// TIA Portal project "trafficLight_timer_counter" (V16)

(* hardware
DEVICE "S7-1200 station_1"  S7-1200 Station
   slot 0: "Rack_0"  S7-1200 Rack  Rack  V1.0
   slot 1: "PLC_1"  CPU 1214C DC/DC/DC  6ES7 214-1AG40-0XB0  V4.4
DEVICE "HMI_1"  KTP700 Basic PN
   slot 0: "HMI_1"  KTP700 Basic PN  6AV2 123-2GB03-0AX0  16.0.0.0
   slot 1: "HMI_RT_1"  KTP700 Basic PN  6AV2 123-2GB03-0AX0  16.0.0.0
   slot 5: "HMI_1.IE_CP_1"  PROFINET Interface  16.0.0.0
      slot 1: "PROFINET Interface_1"  PROFINET Interface
         slot 1: "Port_1"  Port
*)

// ===== PLC "PLC_1"  CPU 1214C DC/DC/DC =====

VAR_GLOBAL   // PLC tag table "Default tag table"
   "GREENTON" AT %MD10 : Time;
   "START(1)" AT %Q0.4 : Bool;
   "RED_SEM" AT %Q0.0 : Bool;
   "REDTON" AT %MD18 : Time;
   "GREEN_SEM" AT %Q0.2 : Bool;
   "BLUETON" AT %MD14 : Time;
   "BLUETON_SEM" AT %MD16 : Time;
   "Tag_8" AT %MD22 : Time;
   "Tag_9" AT %I0.0 : Bool;
   "START(2)" AT %I0.1 : Bool;
   "Tag_11" AT %I0.5 : Bool;
   "STOP_SEM" AT %I1.0 : Bool;
   "BLUE_SEM" AT %Q0.1 : Bool;
   "VALVULA" AT %Q0.3 : Bool;
   "START_SEM" AT %I0.4 : Bool;
   "MEMORIA0" AT %M0.0 : Bool;
   "MEMORIA0.1" AT %M0.1 : Bool;
   "Tag_1" AT %M0.2 : Bool;
   "Tag_3" AT %MW50 : Word;
   "STOP" AT %Q1.0 : Bool;
   "value_norm_x1" AT %IW64 : Int;
   "out_norm_x1" AT %MD200 : Real;
   "value_scale_x1" AT %MD100 : Real;
   "PRESION_VALUE_REAL_scalex1" AT %MD104 : Real;
   "Tag_2" AT %IW68 : Int;
   "Tag_4" AT %MW208 : Word;
   "Tag_5" AT %MD208 : Real;
   "Tag_6" AT %MD102 : Real;
   "Tag_10" AT %MD108 : Real;
   "Tag_12" AT %MD112 : Real;
   "GREENTON_SEM" AT %MD12 : Time;
   "REDTON_SEM" AT %MD20 : Time;
END_VAR

// folder: System blocks/Program resources

DATA_BLOCK "TON1"   // DB2
{ S7_Optimized_Access := 'TRUE' }
AUTHOR : Simatic
FAMILY : IEC
NAME : IEC_TMR
VERSION : 1.0
// stored: InstanceOfName IEC_TIMER
"IEC_TIMER"
BEGIN
END_DATA_BLOCK

DATA_BLOCK "TON2"   // DB5
{ S7_Optimized_Access := 'TRUE' }
AUTHOR : Simatic
FAMILY : IEC
NAME : IEC_TMR
VERSION : 1.0
// stored: InstanceOfName IEC_TIMER
"IEC_TIMER"
BEGIN
END_DATA_BLOCK

DATA_BLOCK "CTU1"   // DB8
{ S7_Optimized_Access := 'TRUE' }
AUTHOR : Simatic
FAMILY : IEC
NAME : CNTR
VERSION : 1.0
// stored: InstanceOfName IEC_COUNTER
"IEC_COUNTER"
BEGIN
END_DATA_BLOCK

DATA_BLOCK "TON3"   // DB10
{ S7_Optimized_Access := 'TRUE' }
AUTHOR : Simatic
FAMILY : IEC
NAME : IEC_TMR
VERSION : 1.0
// stored: InstanceOfName IEC_TIMER
"IEC_TIMER"
BEGIN
END_DATA_BLOCK

// folder: (top level)

FUNCTION "SEMAFORO" : Void   // FC2, LAD
{ S7_Optimized_Access := 'TRUE' }
VERSION : 0.1
BEGIN

REGION Network 1
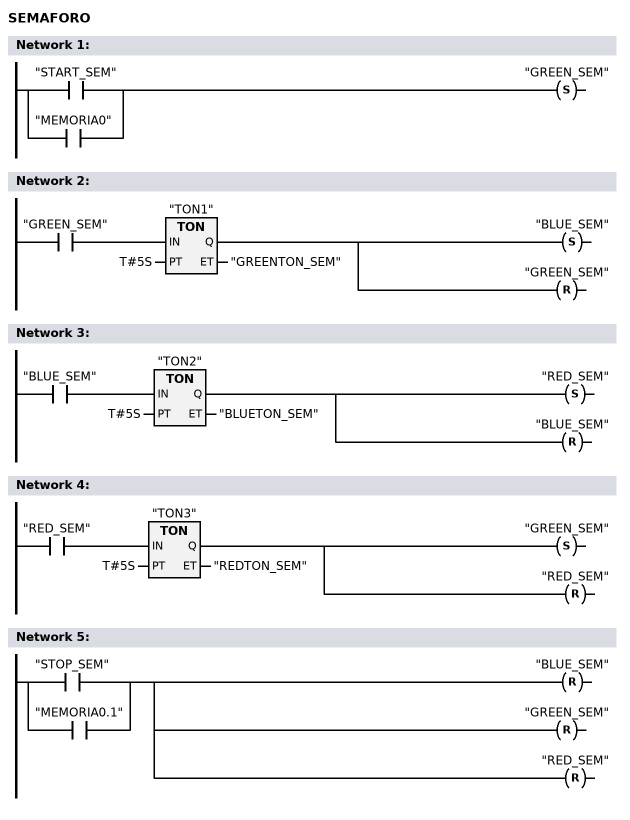
   RUNG wire#powerrail
      Contact( "START_SEM" )
      wire#w1
      S_Coil( "GREEN_SEM" )
   END_RUNG
   RUNG wire#powerrail
      Contact( "MEMORIA0" )
   END_RUNG wire#w1
   // the same network as SCL:
   IF "START_SEM" OR "MEMORIA0" THEN "GREEN_SEM" := TRUE; END_IF;
END_REGION

REGION Network 2
   "TON1".TON(IN := "GREEN_SEM", PT := T#5S, ET => "GREENTON_SEM");
   IF "TON1".Q THEN
       "BLUE_SEM" := TRUE;
       "GREEN_SEM" := FALSE;
   END_IF;
END_REGION

REGION Network 3
   "TON2".TON(IN := "BLUE_SEM", PT := T#5S, ET => "BLUETON_SEM");
   IF "TON2".Q THEN
       "RED_SEM" := TRUE;
       "BLUE_SEM" := FALSE;
   END_IF;
END_REGION

REGION Network 4
   "TON3".TON(IN := "RED_SEM", PT := T#5S, ET => "REDTON_SEM");
   IF "TON3".Q THEN
       "GREEN_SEM" := TRUE;
       "RED_SEM" := FALSE;
   END_IF;
END_REGION

REGION Network 5
   RUNG wire#powerrail
      Contact( "STOP_SEM" )
      wire#w1
      R_Coil( "BLUE_SEM" )
   END_RUNG
   RUNG wire#powerrail
      Contact( "MEMORIA0.1" )
   END_RUNG wire#w1
   RUNG wire#w1
      R_Coil( "GREEN_SEM" )
   END_RUNG
   RUNG wire#w1
      R_Coil( "RED_SEM" )
   END_RUNG
   // the same network as SCL:
   IF "STOP_SEM" OR "MEMORIA0.1" THEN
       "BLUE_SEM" := FALSE;
       "GREEN_SEM" := FALSE;
       "RED_SEM" := FALSE;
   END_IF;
END_REGION
END_FUNCTION

FUNCTION "CONTADOR" : Void   // FC3, LAD
{ S7_Optimized_Access := 'TRUE' }
VERSION : 0.1
   VAR_TEMP   // added for the SCL form of the ladder/FBD networks
      _w1 : Bool;
   END_VAR
BEGIN

REGION Network 1: CONTADOR CTU SIMPLE CON FLANCO DE BAJADA
   // PROHIBICION DE PARTNER OBJECT ELECCION EN SUS PARAMETROS : en memory N item
   // LIMITES CANTIDAD DE ELECCION EN SUS PARAMETROS
   // N ES DE FLANCO DE BAJADAAA
   // si pv = 3, el contador empieza en 0 y se incrementa de 1 en 1 hasta llegar a 3
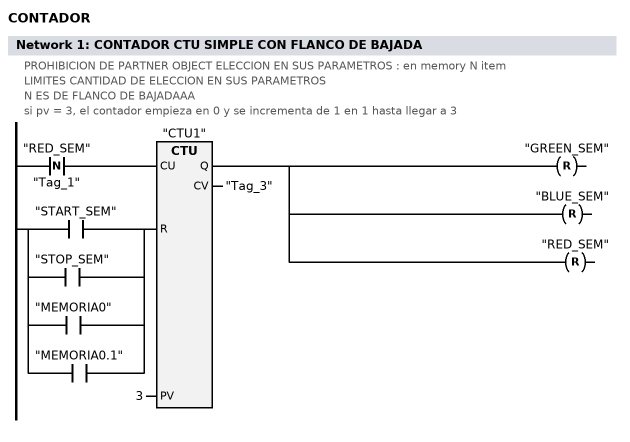
   #_w1 := NOT "RED_SEM" AND "Tag_1";   // falling edge of "RED_SEM"
   "Tag_1" := "RED_SEM";
   "CTU1".CTU(CU := #_w1, R := "START_SEM" OR "STOP_SEM" OR "MEMORIA0" OR "MEMORIA0.1", PV := 3, CV => "Tag_3");
   IF "CTU1".Q THEN
       "GREEN_SEM" := FALSE;
       "BLUE_SEM" := FALSE;
       "RED_SEM" := FALSE;
   END_IF;
END_REGION
END_FUNCTION

ORGANIZATION_BLOCK "Main"   // OB1, LAD, ProgramCycle
TITLE = "Main Program Sweep (Cycle)"
{ S7_Optimized_Access := 'TRUE' }
VERSION : 0.1
   VAR_INPUT
      Initial_Call : Bool;   // Initial call of this OB
      Remanence : Bool;   // =True, if remanent data are available
   END_VAR
BEGIN

REGION Network 1
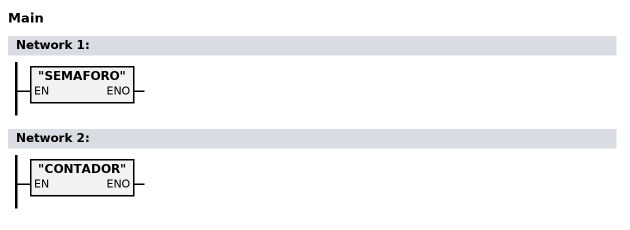
   RUNG wire#powerrail
      "SEMAFORO"()
   END_RUNG
   // the same network as SCL:
   "SEMAFORO"();
END_REGION

REGION Network 2
   RUNG wire#powerrail
      "CONTADOR"()
   END_RUNG
   // the same network as SCL:
   "CONTADOR"();
END_REGION
END_ORGANIZATION_BLOCK

(* ===== HMI "HMI_RT_1" =====
system functions are stored by id; their names below are inferred from use
connection "HMI_Connection_1": ETHERNET, SMART_S7_1200_OMS

HMI tags "Default tag table"
   "Tag_ScreenNumber" : UInt, internal
   "GREEN_SEM" : Bool = PLC GREEN_SEM AT %Q0.2, 1 s
   "BLUE_SEM" : Bool = PLC BLUE_SEM AT %Q0.1, 1 s
   "VALVULA" : Bool = PLC VALVULA AT %Q0.3, 1 s
   "START_SEM" : Bool = PLC START_SEM AT %I0.4, 1 s
   "MEMORIA0" : Bool = PLC MEMORIA0 AT %M0.0, 1 s
   "MEMORIA0.1" : Bool = PLC "MEMORIA0.1" AT %M0.1, 1 s
   "GREENTON" : Time = PLC GREENTON AT %MD10, 1 s
   "BLUETON" : Time = PLC BLUETON AT %MD14, 1 s
   "REDTON" : Time = PLC REDTON AT %MD18, 1 s
   "RED_SEM" : Bool = PLC RED_SEM AT %Q0.0, 1 s
   "GREENTON_SEM" : Time = PLC GREENTON_SEM AT %MD12, 1 s
   "BLUETON_SEM" : Time = PLC BLUETON_SEM AT %MD16, 1 s
   "REDTON_SEM" : Time = PLC REDTON_SEM AT %MD20, 1 s

Template "Template_1" 800x480
   Button "Exit" at 714,429 size 71x50; TextOff 'Exit'; PictureOff "ExitRuntime_KTP700_Basic_PN_TR"; PictureOn "ExitRuntime_KTP700_Basic_PN_TR"
      on Release: StopRuntime(0)
   Button "Template_Button" at 614,429 size 71x50; TextOff 'Text'
   Button "Template_Button_1" at 514,429 size 71x50; TextOff 'Text'
   Button "Template_Button_2" at 414,429 size 71x50; TextOff 'Text'
   Button "Template_Button_3" at 314,429 size 71x50; TextOff 'Text'
   Button "Template_Button_4" at 214,429 size 71x50; TextOff 'Text'
   Button "Template_Button_5" at 114,429 size 71x50; TextOff 'Text'
   Button "Start screen" at 14,429 size 71x50; TextOff 'Start screen'; PictureOff "NavigateHome_KTP700_Basic_PN_TR"; PictureOn "NavigateHome_KTP700_Basic_PN_TR"
      on Release: ActivateScreen("Root screen", 0)
   SymbolicIOField "Symbolic_IO_Field_Screen" at 93,9 size 600x33; TextOff '0'; TextOn '1'; TextList "TextList_ScreenNames"
      ProcessValue <- "Tag_ScreenNumber"
      on Change: ActivateScreenByNumber("Tag_ScreenNumber", 0)
   DateTimeField "HmiScreenItemData" at 695,25 size 105x25
   DateTimeField "HmiScreenItemData_1" at 695,0 size 105x25
   GraphicView "Logo" at 0,0 size 91x51; Picture "Logo of HMI_1"

screen "Root screen" 800x480, template "Template_1"
   on GenerateScreen: SetTag("Tag_ScreenNumber", 1)
   Circle "Circle_1" at 339,208 size 48x48
      Appearance <- "GREEN_SEM"
   Circle "Circle_2" at 337,284 size 48x48
      Appearance <- "BLUE_SEM"
   Circle "Circle_3" at 337,360 size 48x48
      Appearance <- "RED_SEM"
   Button "Button_1" at 535,211 size 96x32; TextOff 'START'
      on Press: SetBit("MEMORIA0")
      on Release: InvertBit("MEMORIA0")
   Button "Button_2" at 537,301 size 96x32; TextOff 'STOP'
      on Press: SetBit("MEMORIA0.1")
      on Release: InvertBit("MEMORIA0.1")
   IOField "I/O field_1" at 413,210 size 96x32; FormatPattern 99999
      ProcessValue <- "GREENTON_SEM"
   TextField "Text field_1" at 255,220 size 61x23; Text 'GREEN'
   TextField "Text field_2" at 266,293 size 47x23; Text 'BLUE'
   TextField "Text field_3" at 273,368 size 39x23; Text 'RED'
   TextField "Text field_4" at 402,176 size 87x23; Text 'TON TIME'
   IOField "I/O field_2" at 413,294 size 96x32; FormatPattern 99999
      ProcessValue <- "BLUETON_SEM"
   IOField "I/O field_3" at 410,372 size 96x32; FormatPattern 99999
      ProcessValue <- "REDTON_SEM"
   TextField "Text field_5" at 530,168 size 184x42; Text 'events - memory 0.0 - press and release'
   TextField "Text field_6" at 535,257 size 232x42; Text 'events - memory 0.0 - press and release'

screen "Screen_1" 800x480
   GraphicView "Graphic view_1" at 508,29 size 82x96; Picture "Graphic_2"
      Visibility <- "VALVULA"
*)